PROGRAM timer1s
VAR
END_VAR

gvl.timer1sec := NOT(gvl.timer1sec);

END_PROGRAM

(* stored: Version 1.1.0.1, ProductVersion 3.1.4024.12
   POU timer1s: Id {33517a13-91ab-46a7-9013-31406b7cb4ca}, SpecialFunc None *)
